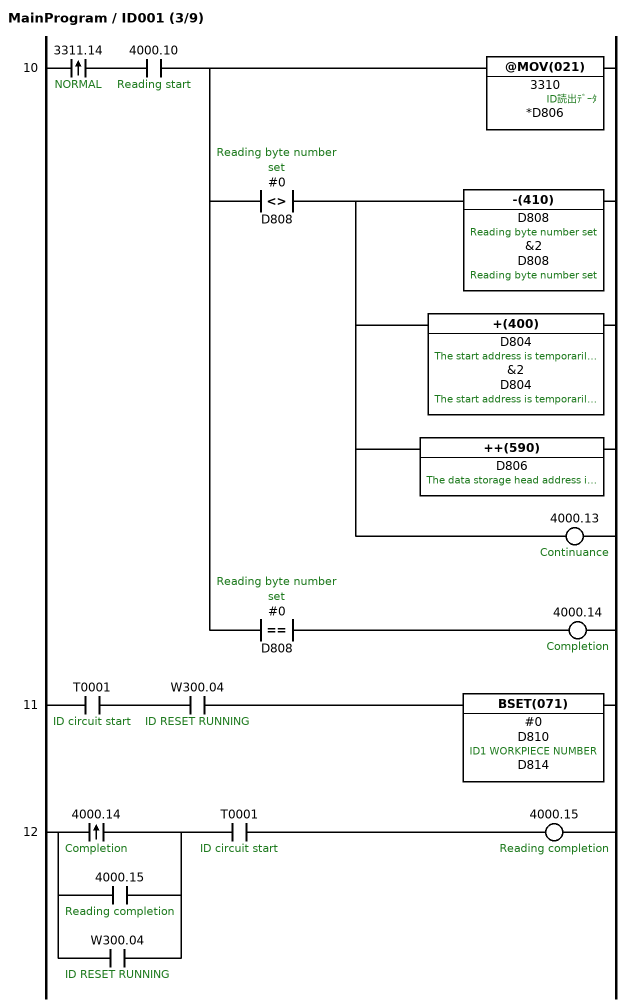
; [picture p24: MainProgram / ID001, rungs 10-12]
; rung 10
@LD 3311.14  ; NORMAL
AND 4000.10  ; Reading start
OUT TR0
@MOV(021) 3310 *D806  ; ID読出ﾃﾞｰﾀ
AND<>(305) #0 D808  ; Reading byte number set
-(410) D808 &2 D808  ; Reading byte number set
+(400) D804 &2 D804  ; The start address is temporarily memorized
++(590) D806  ; The data storage head address is memorized
OUT 4000.13  ; Continuance
LD TR0
AND=(300) #0 D808  ; Reading byte number set
OUT 4000.14  ; Completion
; rung 11
LD T0001  ; ID circuit start
AND W300.04  ; ID RESET RUNNING
BSET(071) #0 D810 D814  ; ID1 WORKPIECE NUMBER
; rung 12
@LD 4000.14  ; Completion
OR 4000.15  ; Reading completion
OR W300.04  ; ID RESET RUNNING
AND T0001  ; ID circuit start
OUT 4000.15  ; Reading completion

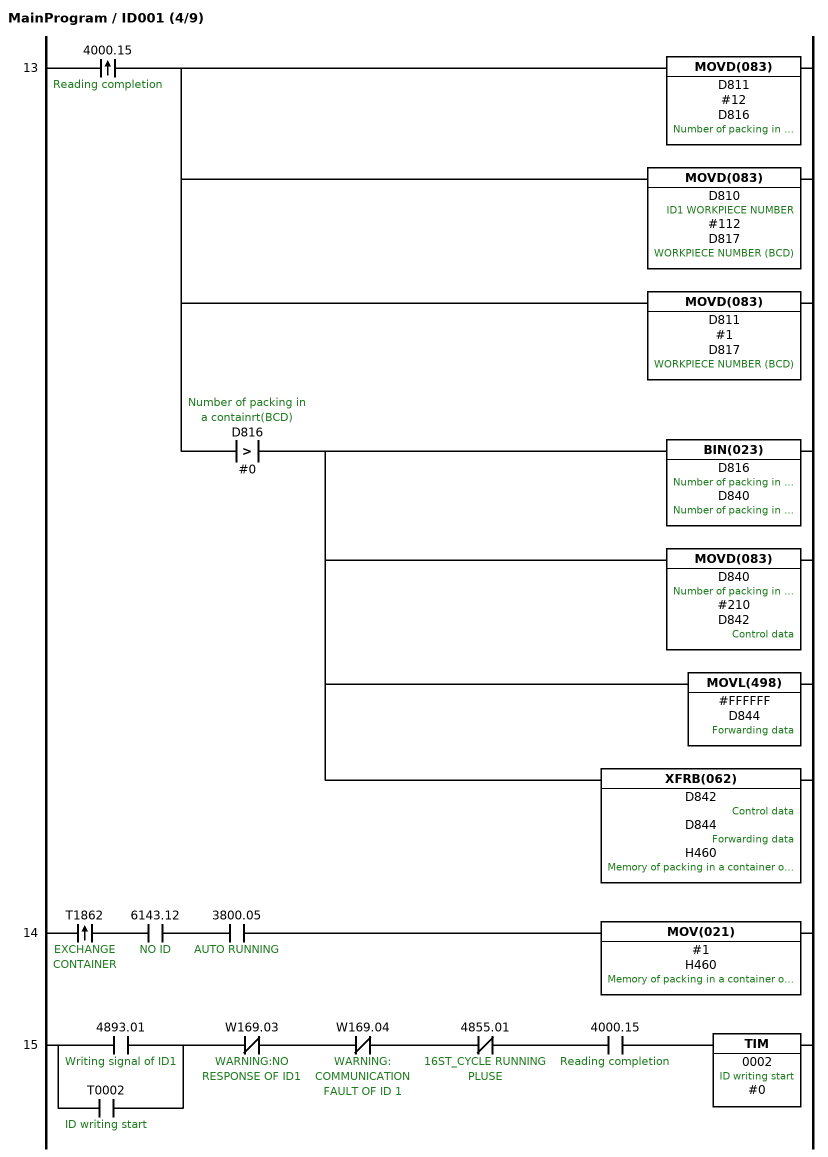
; rung 13
@LD 4000.15  ; Reading completion
MOVD(083) D811 #12 D816  ; Number of packing in a containrt(BCD)
MOVD(083) D810 #112 D817  ; ID1 WORKPIECE NUMBER, WORKPIECE NUMBER (BCD)
MOVD(083) D811 #1 D817  ; WORKPIECE NUMBER (BCD)
AND>(320) D816 #0  ; Number of packing in a containrt(BCD)
BIN(023) D816 D840  ; Number of packing in a containrt(BCD), Number of packing in a containrt(BIN)
MOVD(083) D840 #210 D842  ; Number of packing in a containrt(BIN), Control data
MOVL(498) #FFFFFF D844  ; Forwarding data
XFRB(062) D842 D844 H460  ; Control data, Forwarding data, Memory of packing in a container of lane 1 (exchange container)
; rung 14
@LD T1862  ; EXCHANGE CONTAINER
AND 6143.12  ; NO ID
AND 3800.05  ; AUTO RUNNING
MOV(021) #1 H460  ; Memory of packing in a container of lane 1 (exchange container)
; rung 15
LD 4893.01  ; Writing signal of ID1
OR T0002  ; ID writing start
ANDNOT W169.03  ; WARNING:NO RESPONSE OF ID1
ANDNOT W169.04  ; WARNING:COMMUNICATION FAULT OF ID 1
ANDNOT 4855.01  ; 16ST_CYCLE RUNNING PLUSE
AND 4000.15  ; Reading completion
TIM 0002 #0  ; ID writing start

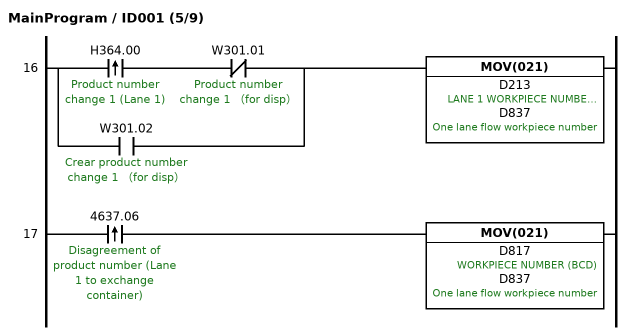
; rung 16
@LD H364.00  ; Product number change 1 (Lane 1)
ANDNOT W301.01  ; Product number change 1 （for disp）
OR W301.02  ; Crear product number change 1 （for disp）
MOV(021) D213 D837  ; LANE 1 WORKPIECE NUMBER DISPLAY, One lane flow workpiece number
; rung 17
@LD 4637.06  ; Disagreement of product number (Lane 1 to exchange container)
MOV(021) D817 D837  ; WORKPIECE NUMBER (BCD), One lane flow workpiece number

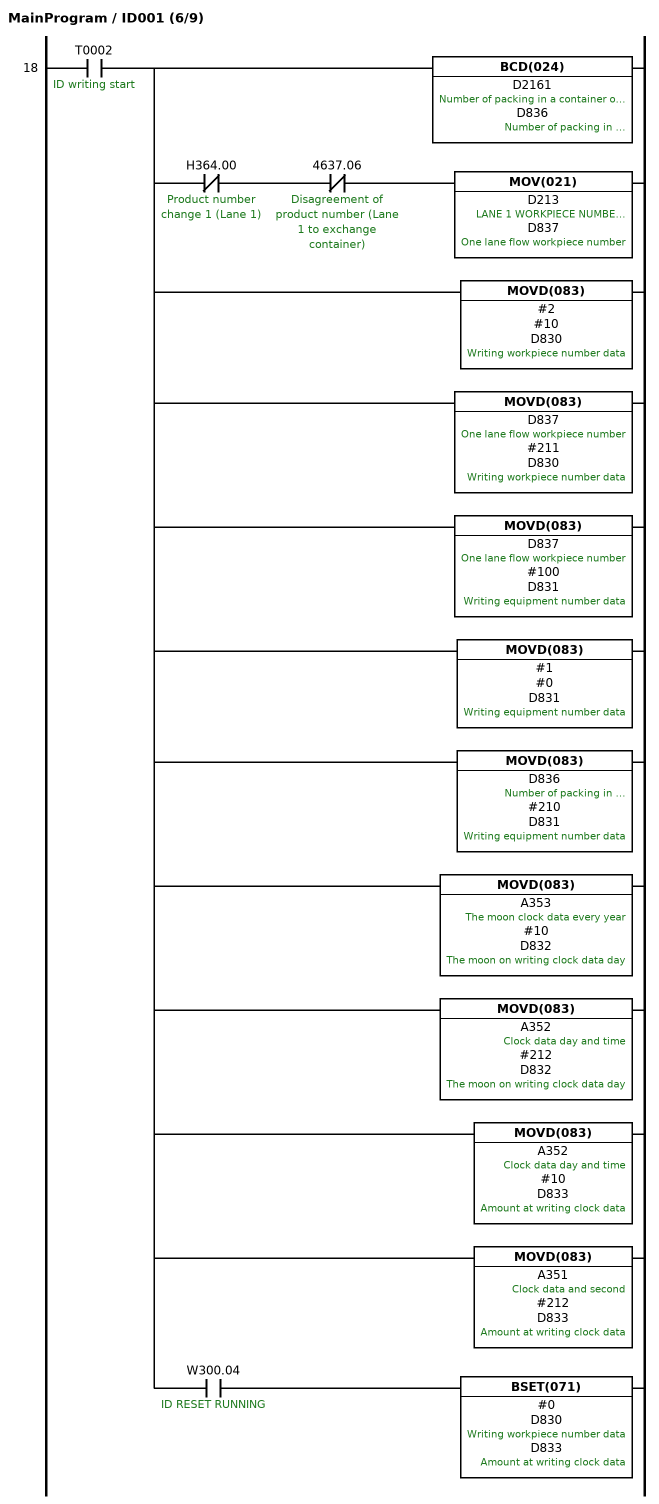
; rung 18
LD T0002  ; ID writing start
OUT TR0
BCD(024) D2161 D836  ; Number of packing in a container of lane 1 (exchange container)(BIN), Number of packing in a containrt(BCD)
ANDNOT H364.00  ; Product number change 1 (Lane 1)
ANDNOT 4637.06  ; Disagreement of product number (Lane 1 to exchange container)
MOV(021) D213 D837  ; LANE 1 WORKPIECE NUMBER DISPLAY, One lane flow workpiece number
LD TR0
MOVD(083) #2 #10 D830  ; Writing workpiece number data
MOVD(083) D837 #211 D830  ; One lane flow workpiece number, Writing workpiece number data
MOVD(083) D837 #100 D831  ; One lane flow workpiece number, Writing equipment number data
MOVD(083) #1 #0 D831  ; Writing equipment number data
MOVD(083) D836 #210 D831  ; Number of packing in a containrt(BCD), Writing equipment number data
MOVD(083) A353 #10 D832  ; The moon clock data every year, The moon on writing clock data day
MOVD(083) A352 #212 D832  ; Clock data day and time, The moon on writing clock data day
MOVD(083) A352 #10 D833  ; Clock data day and time, Amount at writing clock data
MOVD(083) A351 #212 D833  ; Clock data and second, Amount at writing clock data
AND W300.04  ; ID RESET RUNNING
BSET(071) #0 D830 D833  ; Writing workpiece number data, Amount at writing clock data

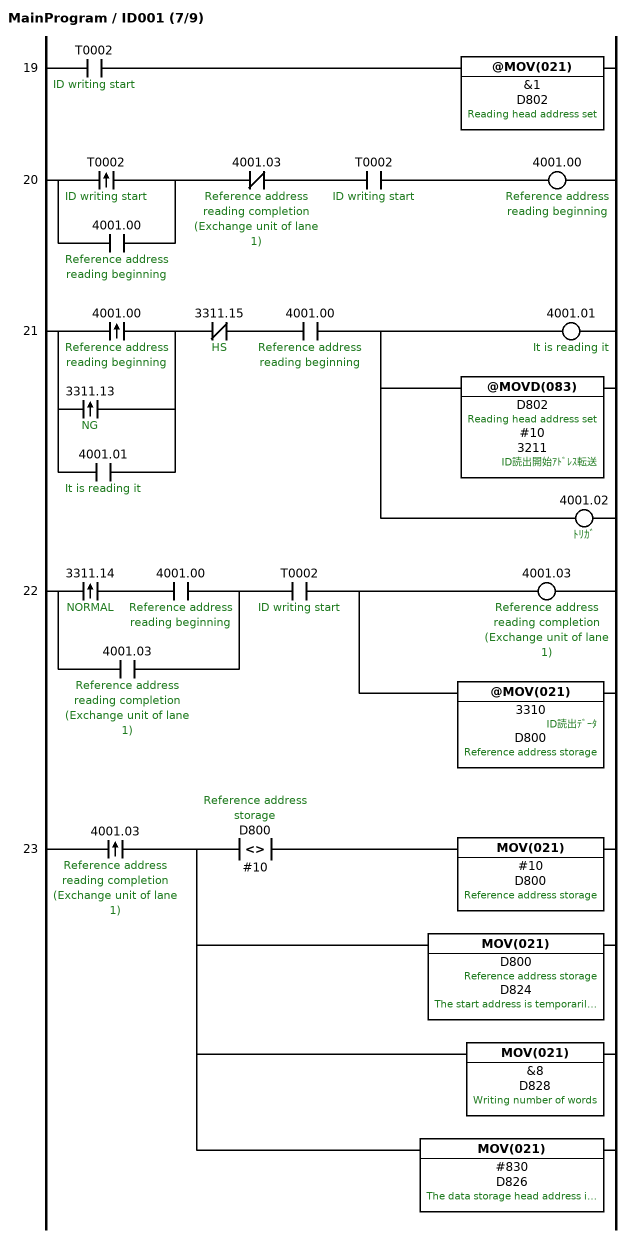
; rung 19
LD T0002  ; ID writing start
@MOV(021) &1 D802  ; Reading head address set
; rung 20
@LD T0002  ; ID writing start
OR 4001.00  ; Reference address reading beginning
ANDNOT 4001.03  ; Reference address reading completion (Exchange unit of lane 1)
AND T0002  ; ID writing start
OUT 4001.00  ; Reference address reading beginning
; rung 21
@LD 4001.00  ; Reference address reading beginning
@OR 3311.13  ; NG
OR 4001.01  ; It is reading it
ANDNOT 3311.15  ; HS
AND 4001.00  ; Reference address reading beginning
OUT 4001.01  ; It is reading it
@MOVD(083) D802 #10 3211  ; Reading head address set, ID読出開始ｱﾄﾞﾚｽ転送
OUT 4001.02  ; ﾄﾘｶﾞ
; rung 22
@LD 3311.14  ; NORMAL
AND 4001.00  ; Reference address reading beginning
OR 4001.03  ; Reference address reading completion (Exchange unit of lane 1)
AND T0002  ; ID writing start
OUT 4001.03  ; Reference address reading completion (Exchange unit of lane 1)
@MOV(021) 3310 D800  ; ID読出ﾃﾞｰﾀ, Reference address storage
; rung 23
@LD 4001.03  ; Reference address reading completion (Exchange unit of lane 1)
OUT TR0
AND<>(305) D800 #10  ; Reference address storage
MOV(021) #10 D800  ; Reference address storage
LD TR0
MOV(021) D800 D824  ; Reference address storage, The start address is temporarily memorized
MOV(021) &8 D828  ; Writing number of words
MOV(021) #830 D826  ; The data storage head address is memorized

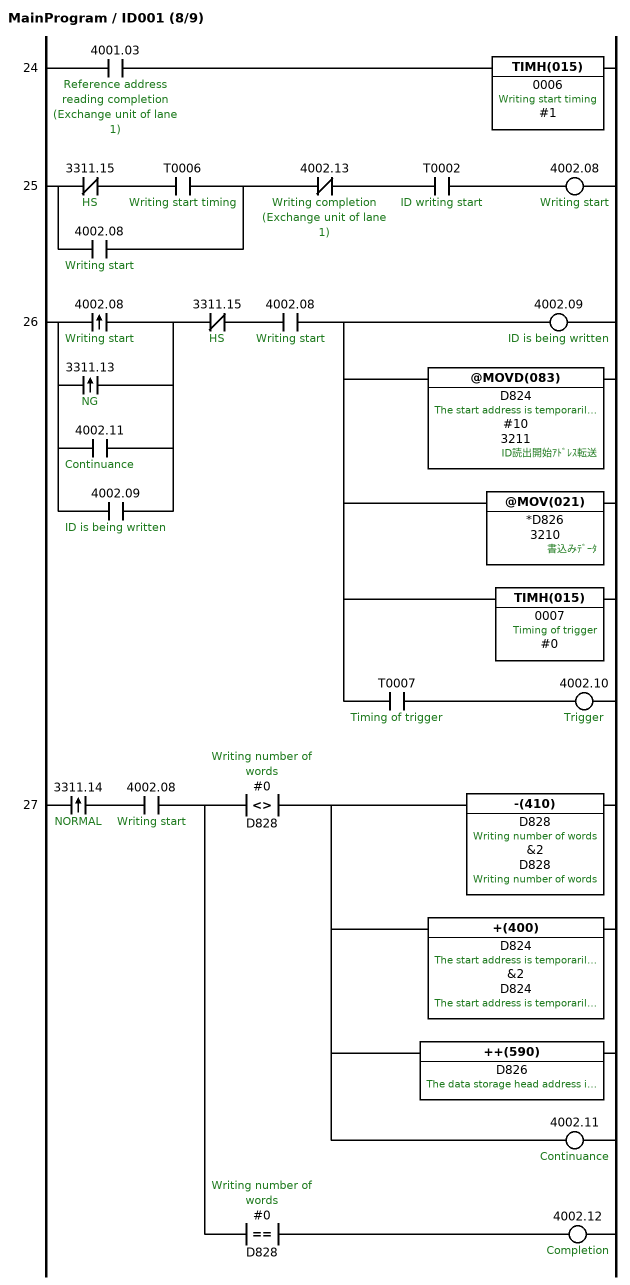
; rung 24
LD 4001.03  ; Reference address reading completion (Exchange unit of lane 1)
TIMH(015) 0006 #1  ; Writing start timing
; rung 25
LDNOT 3311.15  ; HS
AND T0006  ; Writing start timing
OR 4002.08  ; Writing start
ANDNOT 4002.13  ; Writing completion (Exchange unit of lane 1)
AND T0002  ; ID writing start
OUT 4002.08  ; Writing start
; rung 26
@LD 4002.08  ; Writing start
@OR 3311.13  ; NG
OR 4002.11  ; Continuance
OR 4002.09  ; ID is being written
ANDNOT 3311.15  ; HS
AND 4002.08  ; Writing start
OUT 4002.09  ; ID is being written
@MOVD(083) D824 #10 3211  ; The start address is temporarily memorized, ID読出開始ｱﾄﾞﾚｽ転送
@MOV(021) *D826 3210  ; 書込みﾃﾞｰﾀ
TIMH(015) 0007 #0  ; Timing of trigger
AND T0007  ; Timing of trigger
OUT 4002.10  ; Trigger
; rung 27
@LD 3311.14  ; NORMAL
AND 4002.08  ; Writing start
OUT TR0
AND<>(305) #0 D828  ; Writing number of words
-(410) D828 &2 D828  ; Writing number of words
+(400) D824 &2 D824  ; The start address is temporarily memorized
++(590) D826  ; The data storage head address is memorized
OUT 4002.11  ; Continuance
LD TR0
AND=(300) #0 D828  ; Writing number of words
OUT 4002.12  ; Completion

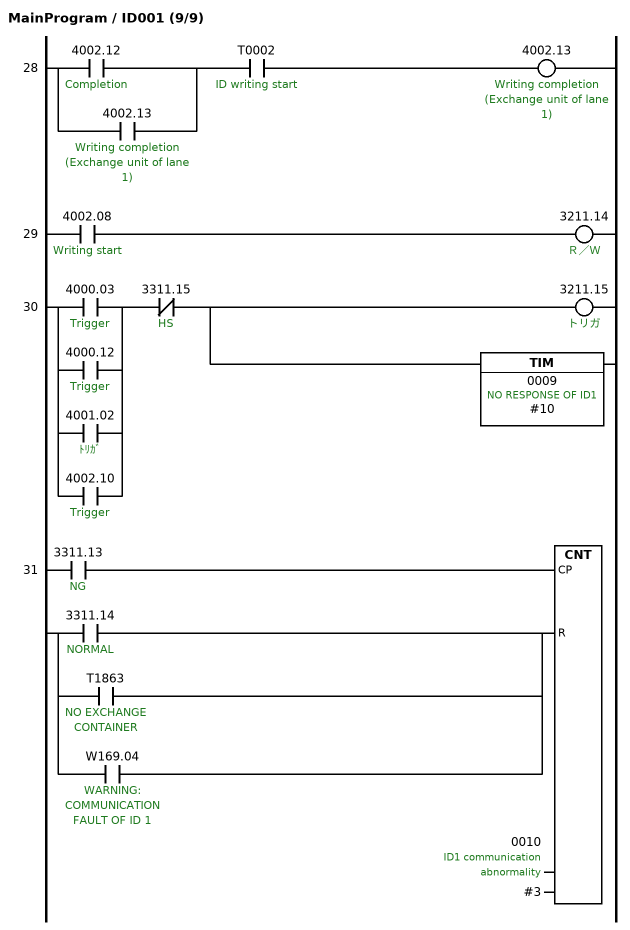
; rung 28
LD 4002.12  ; Completion
OR 4002.13  ; Writing completion (Exchange unit of lane 1)
AND T0002  ; ID writing start
OUT 4002.13  ; Writing completion (Exchange unit of lane 1)
; rung 29
LD 4002.08  ; Writing start
OUT 3211.14  ; Ｒ／Ｗ
; rung 30
LD 4000.03  ; Trigger
OR 4000.12  ; Trigger
OR 4001.02  ; ﾄﾘｶﾞ
OR 4002.10  ; Trigger
ANDNOT 3311.15  ; HS
OUT 3211.15  ; トリガ
TIM 0009 #10  ; NO RESPONSE OF ID1
; rung 31
LD 3311.13  ; NG
LD 3311.14  ; NORMAL
OR T1863  ; NO EXCHANGE CONTAINER
OR W169.04  ; WARNING:COMMUNICATION FAULT OF ID 1
CNT 0010 #3  ; ID1 communication abnormality

### Section ID002

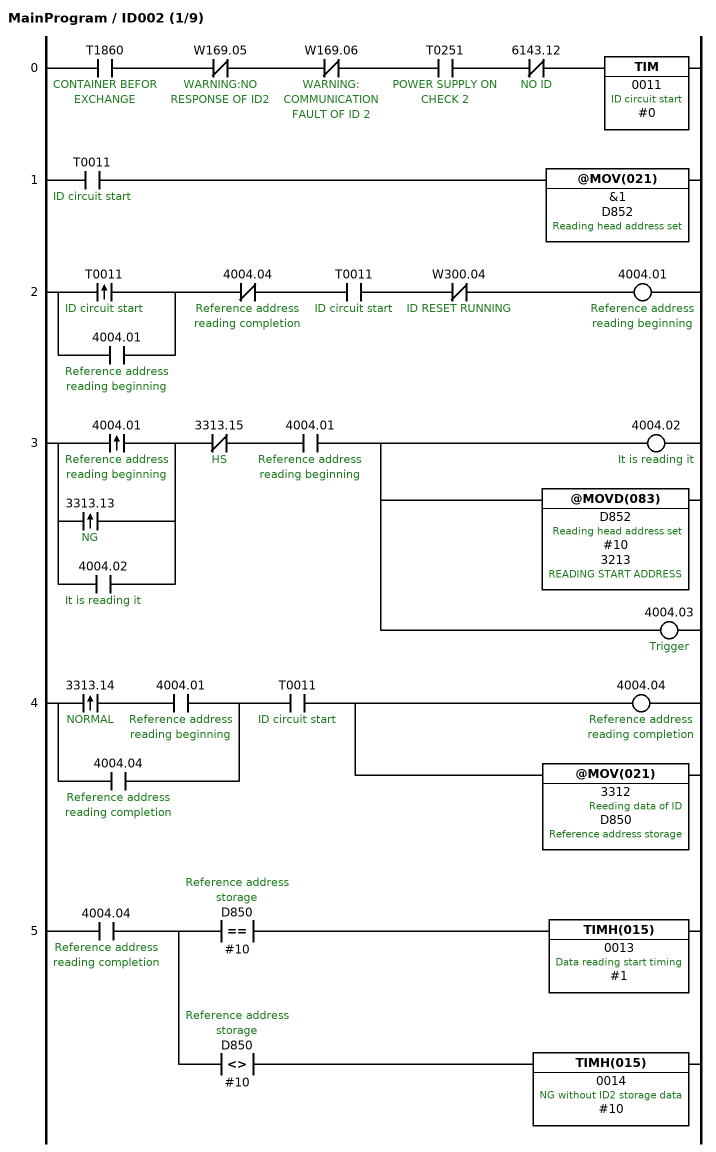
; rung 0
LD T1860  ; CONTAINER BEFOR EXCHANGE
ANDNOT W169.05  ; WARNING:NO RESPONSE OF ID2
ANDNOT W169.06  ; WARNING:COMMUNICATION FAULT OF ID 2
AND T0251  ; POWER SUPPLY ON CHECK 2
ANDNOT 6143.12  ; NO ID
TIM 0011 #0  ; ID circuit start
; rung 1
LD T0011  ; ID circuit start
@MOV(021) &1 D852  ; Reading head address set
; rung 2
@LD T0011  ; ID circuit start
OR 4004.01  ; Reference address reading beginning
ANDNOT 4004.04  ; Reference address reading completion
AND T0011  ; ID circuit start
ANDNOT W300.04  ; ID RESET RUNNING
OUT 4004.01  ; Reference address reading beginning
; rung 3
@LD 4004.01  ; Reference address reading beginning
@OR 3313.13  ; NG
OR 4004.02  ; It is reading it
ANDNOT 3313.15  ; HS
AND 4004.01  ; Reference address reading beginning
OUT 4004.02  ; It is reading it
@MOVD(083) D852 #10 3213  ; Reading head address set, READING START ADDRESS
OUT 4004.03  ; Trigger
; rung 4
@LD 3313.14  ; NORMAL
AND 4004.01  ; Reference address reading beginning
OR 4004.04  ; Reference address reading completion
AND T0011  ; ID circuit start
OUT 4004.04  ; Reference address reading completion
@MOV(021) 3312 D850  ; Reeding data of ID, Reference address storage
; rung 5
LD 4004.04  ; Reference address reading completion
OUT TR0
AND=(300) D850 #10  ; Reference address storage
TIMH(015) 0013 #1  ; Data reading start timing
LD TR0
AND<>(305) D850 #10  ; Reference address storage
TIMH(015) 0014 #10  ; NG without ID2 storage data

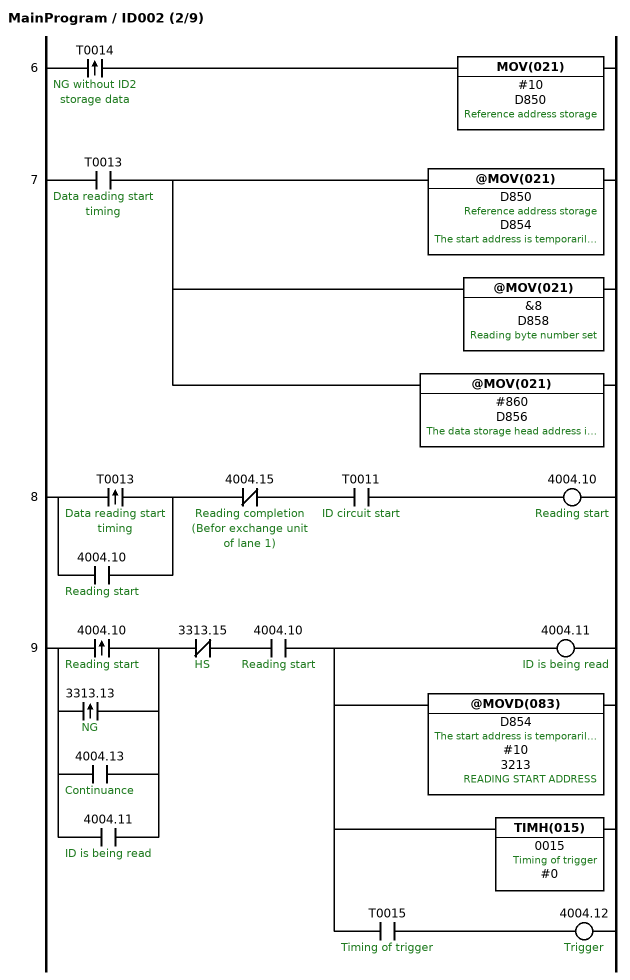
; rung 6
@LD T0014  ; NG without ID2 storage data
MOV(021) #10 D850  ; Reference address storage
; rung 7
LD T0013  ; Data reading start timing
@MOV(021) D850 D854  ; Reference address storage, The start address is temporarily memorized
@MOV(021) &8 D858  ; Reading byte number set
@MOV(021) #860 D856  ; The data storage head address is memorized
; rung 8
@LD T0013  ; Data reading start timing
OR 4004.10  ; Reading start
ANDNOT 4004.15  ; Reading completion (Befor exchange unit of lane 1)
AND T0011  ; ID circuit start
OUT 4004.10  ; Reading start
; rung 9
@LD 4004.10  ; Reading start
@OR 3313.13  ; NG
OR 4004.13  ; Continuance
OR 4004.11  ; ID is being read
ANDNOT 3313.15  ; HS
AND 4004.10  ; Reading start
OUT 4004.11  ; ID is being read
@MOVD(083) D854 #10 3213  ; The start address is temporarily memorized, READING START ADDRESS
TIMH(015) 0015 #0  ; Timing of trigger
AND T0015  ; Timing of trigger
OUT 4004.12  ; Trigger

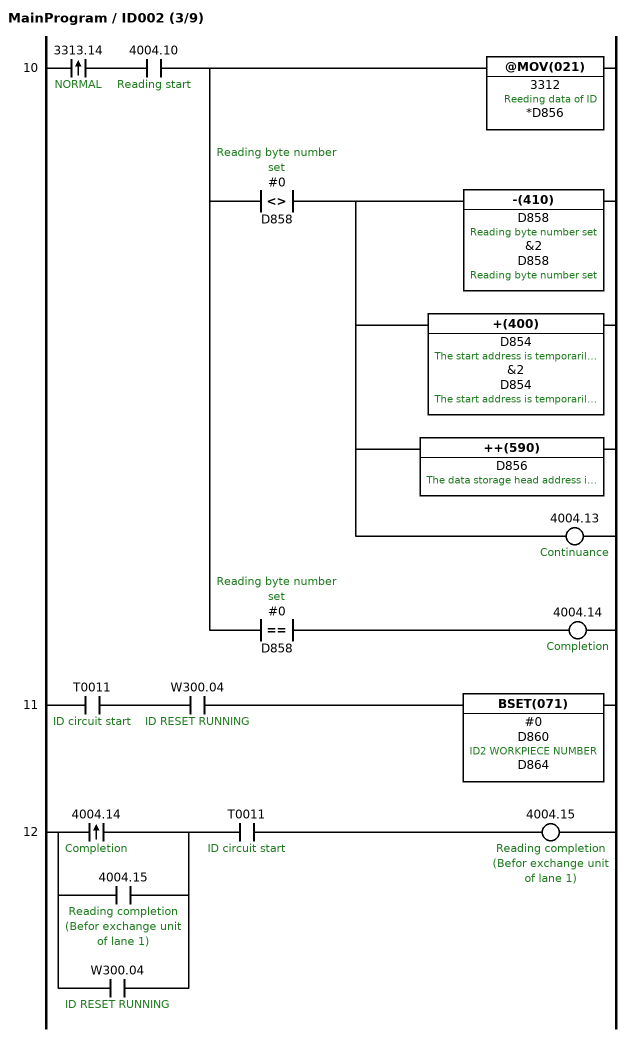
; rung 10
@LD 3313.14  ; NORMAL
AND 4004.10  ; Reading start
OUT TR0
@MOV(021) 3312 *D856  ; Reeding data of ID
AND<>(305) #0 D858  ; Reading byte number set
-(410) D858 &2 D858  ; Reading byte number set
+(400) D854 &2 D854  ; The start address is temporarily memorized
++(590) D856  ; The data storage head address is memorized
OUT 4004.13  ; Continuance
LD TR0
AND=(300) #0 D858  ; Reading byte number set
OUT 4004.14  ; Completion
; rung 11
LD T0011  ; ID circuit start
AND W300.04  ; ID RESET RUNNING
BSET(071) #0 D860 D864  ; ID2 WORKPIECE NUMBER
; rung 12
@LD 4004.14  ; Completion
OR 4004.15  ; Reading completion (Befor exchange unit of lane 1)
OR W300.04  ; ID RESET RUNNING
AND T0011  ; ID circuit start
OUT 4004.15  ; Reading completion (Befor exchange unit of lane 1)

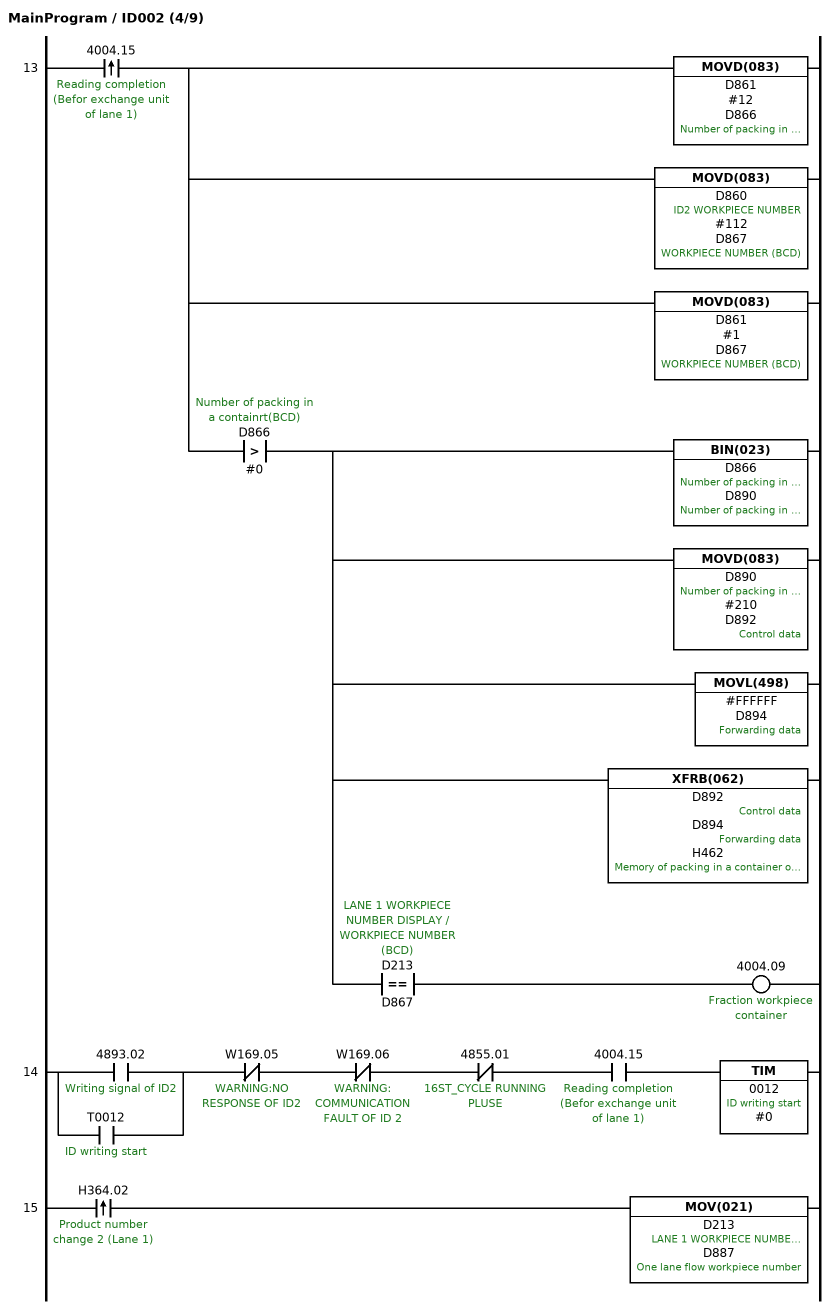
; rung 13
@LD 4004.15  ; Reading completion (Befor exchange unit of lane 1)
MOVD(083) D861 #12 D866  ; Number of packing in a containrt(BCD)
MOVD(083) D860 #112 D867  ; ID2 WORKPIECE NUMBER, WORKPIECE NUMBER (BCD)
MOVD(083) D861 #1 D867  ; WORKPIECE NUMBER (BCD)
AND>(320) D866 #0  ; Number of packing in a containrt(BCD)
BIN(023) D866 D890  ; Number of packing in a containrt(BCD), Number of packing in a containrt(BIN)
MOVD(083) D890 #210 D892  ; Number of packing in a containrt(BIN), Control data
MOVL(498) #FFFFFF D894  ; Forwarding data
XFRB(062) D892 D894 H462  ; Control data, Forwarding data, Memory of packing in a container of lane 1 (container befor exchange)
AND=(300) D213 D867  ; LANE 1 WORKPIECE NUMBER DISPLAY, WORKPIECE NUMBER (BCD)
OUT 4004.09  ; Fraction workpiece container
; rung 14
LD 4893.02  ; Writing signal of ID2
OR T0012  ; ID writing start
ANDNOT W169.05  ; WARNING:NO RESPONSE OF ID2
ANDNOT W169.06  ; WARNING:COMMUNICATION FAULT OF ID 2
ANDNOT 4855.01  ; 16ST_CYCLE RUNNING PLUSE
AND 4004.15  ; Reading completion (Befor exchange unit of lane 1)
TIM 0012 #0  ; ID writing start
; rung 15
@LD H364.02  ; Product number change 2 (Lane 1)
MOV(021) D213 D887  ; LANE 1 WORKPIECE NUMBER DISPLAY, One lane flow workpiece number

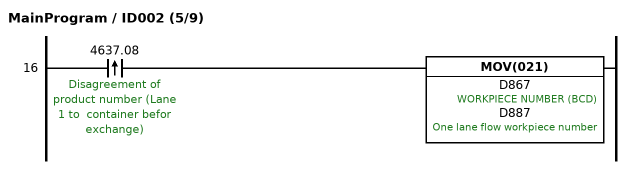
; rung 16
@LD 4637.08  ; Disagreement of product number (Lane 1 to  container befor exchange)
MOV(021) D867 D887  ; WORKPIECE NUMBER (BCD), One lane flow workpiece number

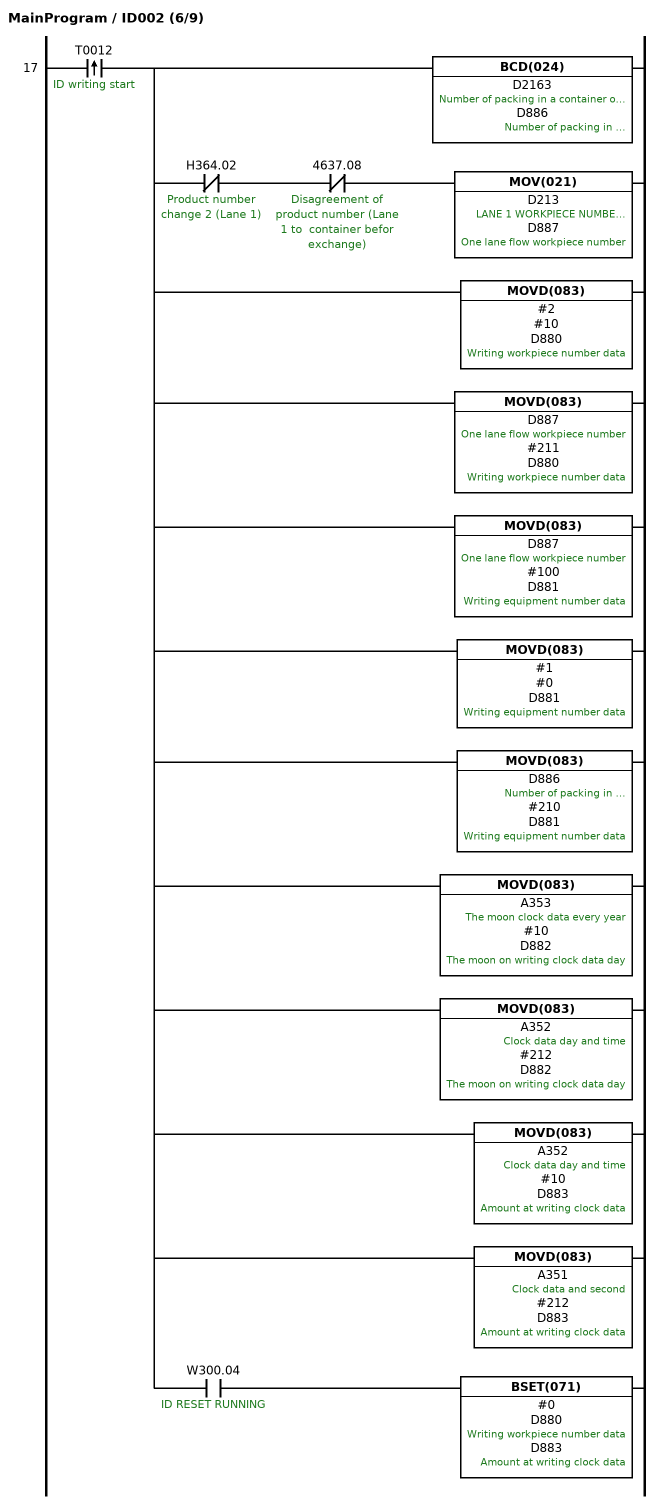
; rung 17
@LD T0012  ; ID writing start
OUT TR0
BCD(024) D2163 D886  ; Number of packing in a container of lane 1 (container before exchange)(BIN), Number of packing in a containrt(BCD)
ANDNOT H364.02  ; Product number change 2 (Lane 1)
ANDNOT 4637.08  ; Disagreement of product number (Lane 1 to  container befor exchange)
MOV(021) D213 D887  ; LANE 1 WORKPIECE NUMBER DISPLAY, One lane flow workpiece number
LD TR0
MOVD(083) #2 #10 D880  ; Writing workpiece number data
MOVD(083) D887 #211 D880  ; One lane flow workpiece number, Writing workpiece number data
MOVD(083) D887 #100 D881  ; One lane flow workpiece number, Writing equipment number data
MOVD(083) #1 #0 D881  ; Writing equipment number data
MOVD(083) D886 #210 D881  ; Number of packing in a containrt(BCD), Writing equipment number data
MOVD(083) A353 #10 D882  ; The moon clock data every year, The moon on writing clock data day
MOVD(083) A352 #212 D882  ; Clock data day and time, The moon on writing clock data day
MOVD(083) A352 #10 D883  ; Clock data day and time, Amount at writing clock data
MOVD(083) A351 #212 D883  ; Clock data and second, Amount at writing clock data
AND W300.04  ; ID RESET RUNNING
BSET(071) #0 D880 D883  ; Writing workpiece number data, Amount at writing clock data

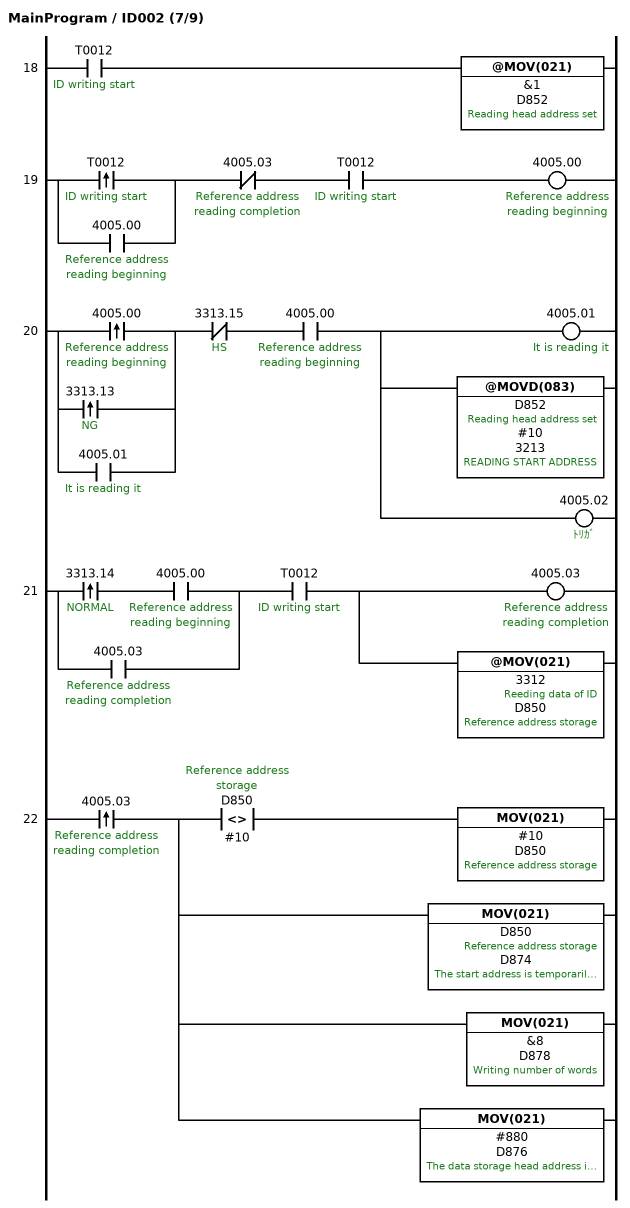
; rung 18
LD T0012  ; ID writing start
@MOV(021) &1 D852  ; Reading head address set
; rung 19
@LD T0012  ; ID writing start
OR 4005.00  ; Reference address reading beginning
ANDNOT 4005.03  ; Reference address reading completion
AND T0012  ; ID writing start
OUT 4005.00  ; Reference address reading beginning
; rung 20
@LD 4005.00  ; Reference address reading beginning
@OR 3313.13  ; NG
OR 4005.01  ; It is reading it
ANDNOT 3313.15  ; HS
AND 4005.00  ; Reference address reading beginning
OUT 4005.01  ; It is reading it
@MOVD(083) D852 #10 3213  ; Reading head address set, READING START ADDRESS
OUT 4005.02  ; ﾄﾘｶﾞ
; rung 21
@LD 3313.14  ; NORMAL
AND 4005.00  ; Reference address reading beginning
OR 4005.03  ; Reference address reading completion
AND T0012  ; ID writing start
OUT 4005.03  ; Reference address reading completion
@MOV(021) 3312 D850  ; Reeding data of ID, Reference address storage
; rung 22
@LD 4005.03  ; Reference address reading completion
OUT TR0
AND<>(305) D850 #10  ; Reference address storage
MOV(021) #10 D850  ; Reference address storage
LD TR0
MOV(021) D850 D874  ; Reference address storage, The start address is temporarily memorized
MOV(021) &8 D878  ; Writing number of words
MOV(021) #880 D876  ; The data storage head address is memorized

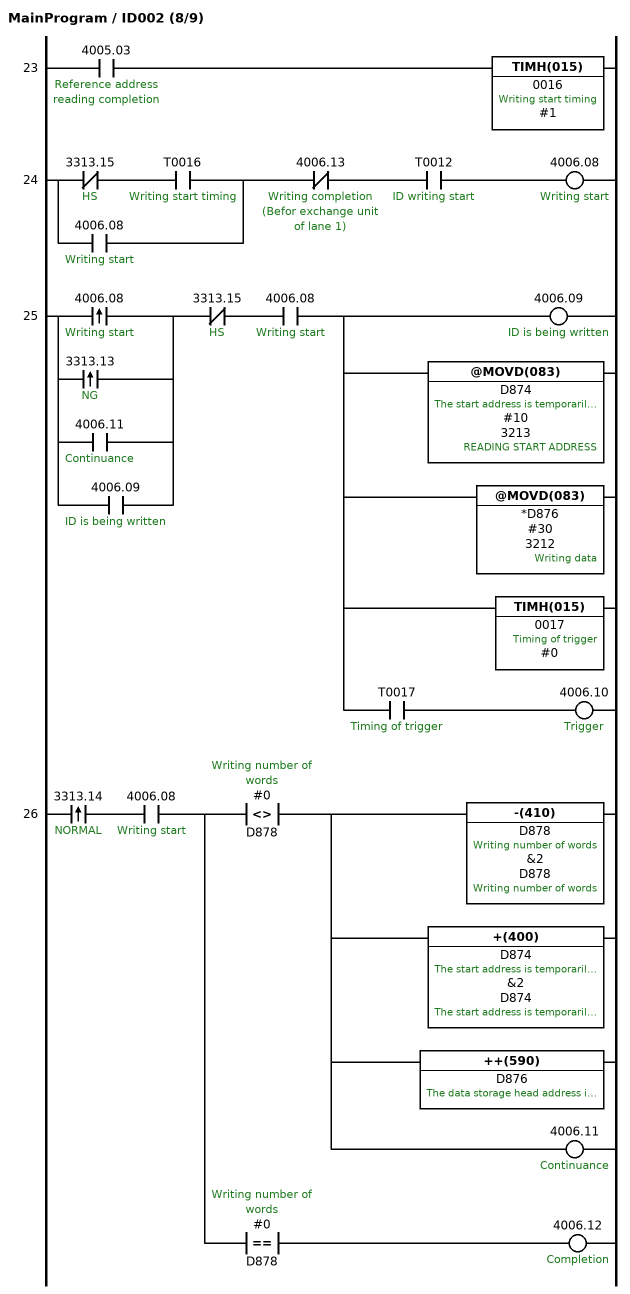
; rung 23
LD 4005.03  ; Reference address reading completion
TIMH(015) 0016 #1  ; Writing start timing
; rung 24
LDNOT 3313.15  ; HS
AND T0016  ; Writing start timing
OR 4006.08  ; Writing start
ANDNOT 4006.13  ; Writing completion (Befor exchange unit of lane 1)
AND T0012  ; ID writing start
OUT 4006.08  ; Writing start
; rung 25
@LD 4006.08  ; Writing start
@OR 3313.13  ; NG
OR 4006.11  ; Continuance
OR 4006.09  ; ID is being written
ANDNOT 3313.15  ; HS
AND 4006.08  ; Writing start
OUT 4006.09  ; ID is being written
@MOVD(083) D874 #10 3213  ; The start address is temporarily memorized, READING START ADDRESS
@MOVD(083) *D876 #30 3212  ; Writing data
TIMH(015) 0017 #0  ; Timing of trigger
AND T0017  ; Timing of trigger
OUT 4006.10  ; Trigger
; rung 26
@LD 3313.14  ; NORMAL
AND 4006.08  ; Writing start
OUT TR0
AND<>(305) #0 D878  ; Writing number of words
-(410) D878 &2 D878  ; Writing number of words
+(400) D874 &2 D874  ; The start address is temporarily memorized
++(590) D876  ; The data storage head address is memorized
OUT 4006.11  ; Continuance
LD TR0
AND=(300) #0 D878  ; Writing number of words
OUT 4006.12  ; Completion

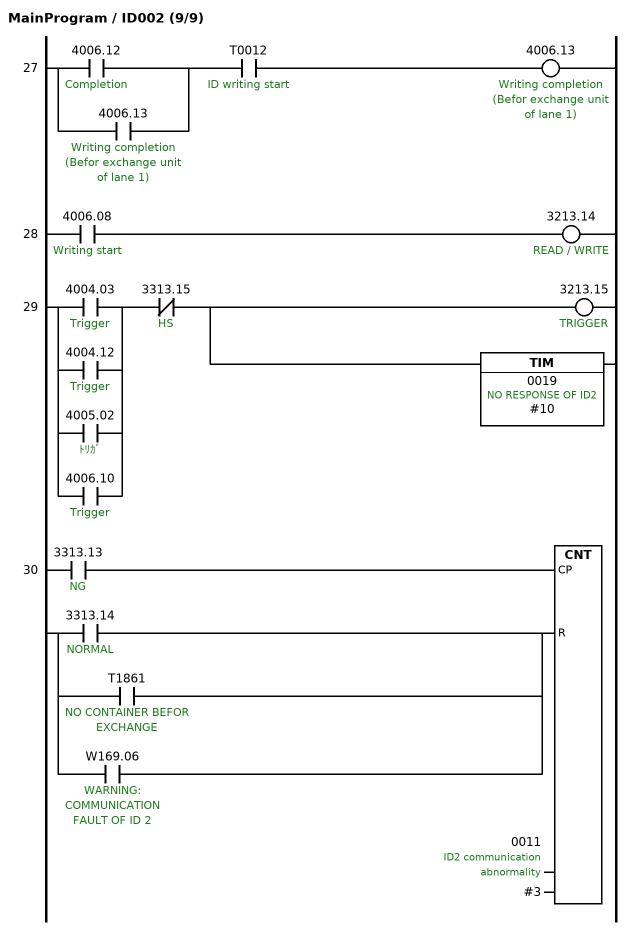
; rung 27
LD 4006.12  ; Completion
OR 4006.13  ; Writing completion (Befor exchange unit of lane 1)
AND T0012  ; ID writing start
OUT 4006.13  ; Writing completion (Befor exchange unit of lane 1)
; rung 28
LD 4006.08  ; Writing start
OUT 3213.14  ; READ / WRITE
; rung 29
LD 4004.03  ; Trigger
OR 4004.12  ; Trigger
OR 4005.02  ; ﾄﾘｶﾞ
OR 4006.10  ; Trigger
ANDNOT 3313.15  ; HS
OUT 3213.15  ; TRIGGER
TIM 0019 #10  ; NO RESPONSE OF ID2
; rung 30
LD 3313.13  ; NG
LD 3313.14  ; NORMAL
OR T1861  ; NO CONTAINER BEFOR EXCHANGE
OR W169.06  ; WARNING:COMMUNICATION FAULT OF ID 2
CNT 0011 #3  ; ID2 communication abnormality

### Section ID003

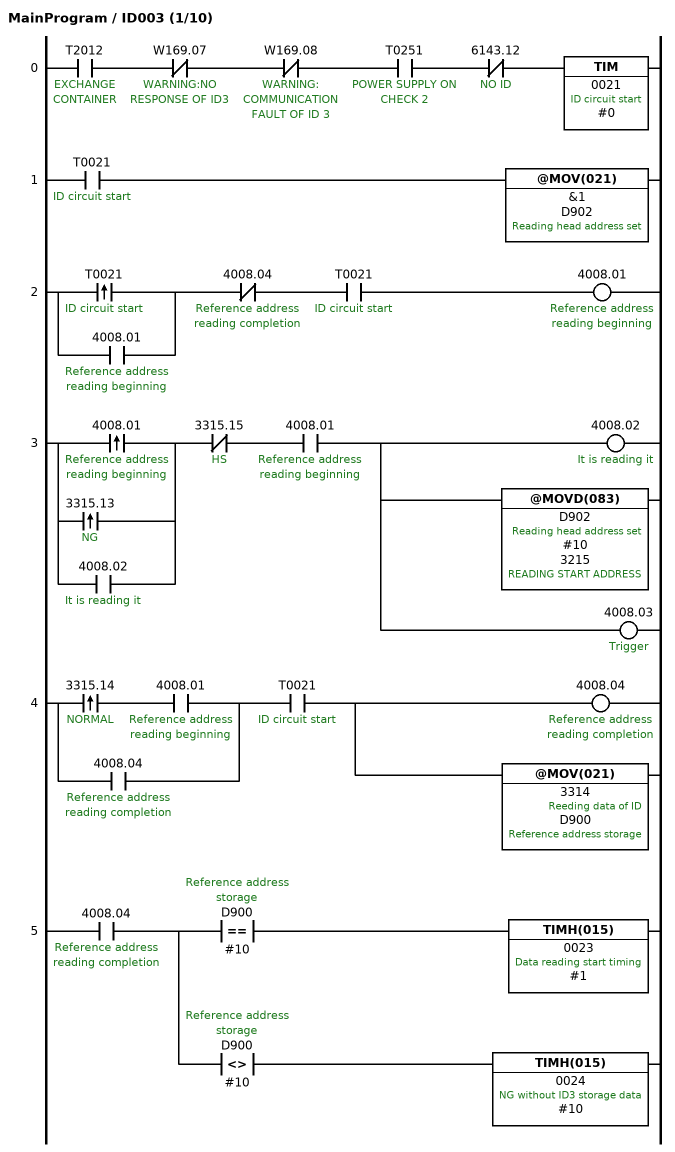
; rung 0
LD T2012  ; EXCHANGE CONTAINER
ANDNOT W169.07  ; WARNING:NO RESPONSE OF ID3
ANDNOT W169.08  ; WARNING:COMMUNICATION FAULT OF ID 3
AND T0251  ; POWER SUPPLY ON CHECK 2
ANDNOT 6143.12  ; NO ID
TIM 0021 #0  ; ID circuit start
; rung 1
LD T0021  ; ID circuit start
@MOV(021) &1 D902  ; Reading head address set
; rung 2
@LD T0021  ; ID circuit start
OR 4008.01  ; Reference address reading beginning
ANDNOT 4008.04  ; Reference address reading completion
AND T0021  ; ID circuit start
OUT 4008.01  ; Reference address reading beginning
; rung 3
@LD 4008.01  ; Reference address reading beginning
@OR 3315.13  ; NG
OR 4008.02  ; It is reading it
ANDNOT 3315.15  ; HS
AND 4008.01  ; Reference address reading beginning
OUT 4008.02  ; It is reading it
@MOVD(083) D902 #10 3215  ; Reading head address set, READING START ADDRESS
OUT 4008.03  ; Trigger
; rung 4
@LD 3315.14  ; NORMAL
AND 4008.01  ; Reference address reading beginning
OR 4008.04  ; Reference address reading completion
AND T0021  ; ID circuit start
OUT 4008.04  ; Reference address reading completion
@MOV(021) 3314 D900  ; Reeding data of ID, Reference address storage
; rung 5
LD 4008.04  ; Reference address reading completion
OUT TR0
AND=(300) D900 #10  ; Reference address storage
TIMH(015) 0023 #1  ; Data reading start timing
LD TR0
AND<>(305) D900 #10  ; Reference address storage
TIMH(015) 0024 #10  ; NG without ID3 storage data

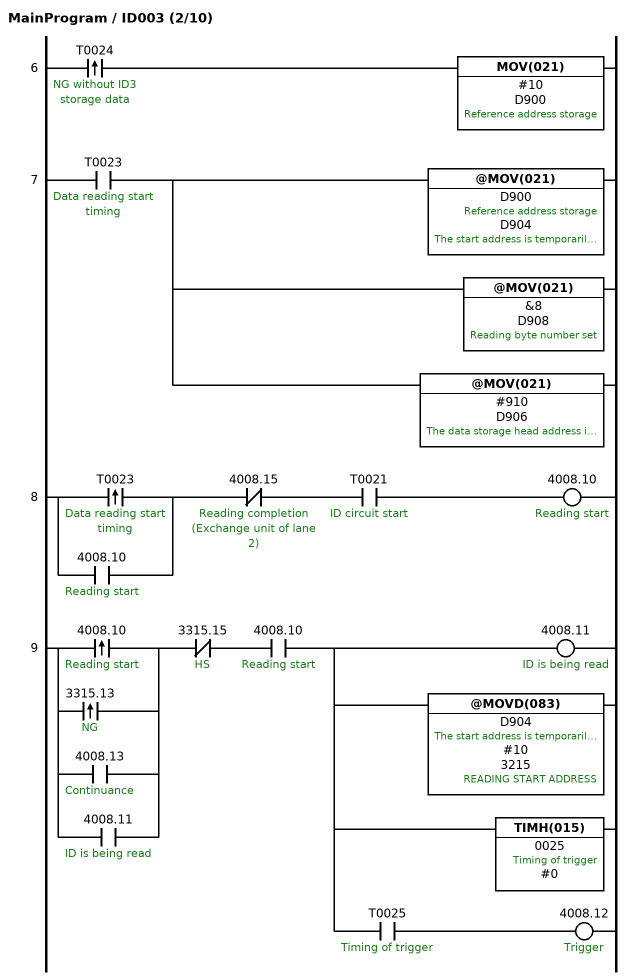
; rung 6
@LD T0024  ; NG without ID3 storage data
MOV(021) #10 D900  ; Reference address storage
; rung 7
LD T0023  ; Data reading start timing
@MOV(021) D900 D904  ; Reference address storage, The start address is temporarily memorized
@MOV(021) &8 D908  ; Reading byte number set
@MOV(021) #910 D906  ; The data storage head address is memorized
; rung 8
@LD T0023  ; Data reading start timing
OR 4008.10  ; Reading start
ANDNOT 4008.15  ; Reading completion (Exchange unit of lane 2)
AND T0021  ; ID circuit start
OUT 4008.10  ; Reading start
; rung 9
@LD 4008.10  ; Reading start
@OR 3315.13  ; NG
OR 4008.13  ; Continuance
OR 4008.11  ; ID is being read
ANDNOT 3315.15  ; HS
AND 4008.10  ; Reading start
OUT 4008.11  ; ID is being read
@MOVD(083) D904 #10 3215  ; The start address is temporarily memorized, READING START ADDRESS
TIMH(015) 0025 #0  ; Timing of trigger
AND T0025  ; Timing of trigger
OUT 4008.12  ; Trigger

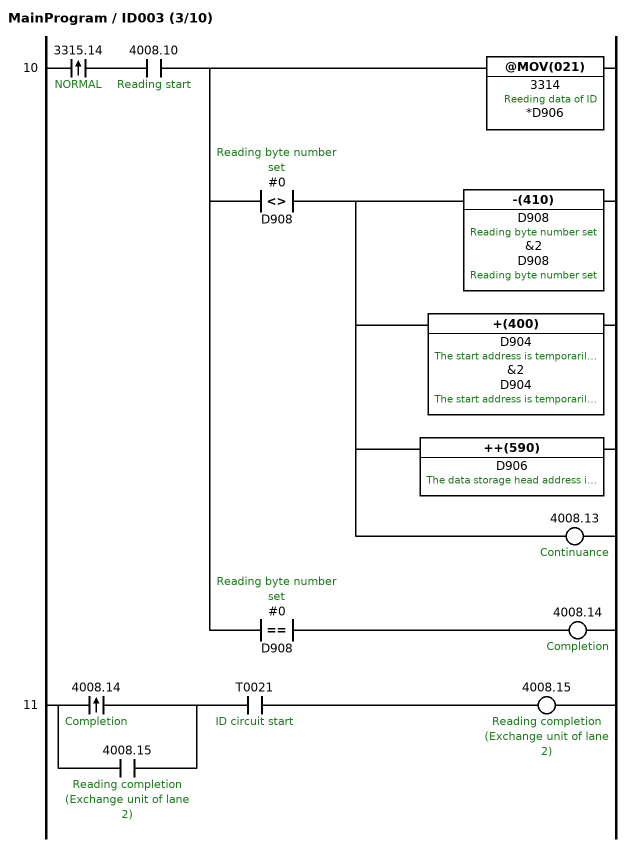
; rung 10
@LD 3315.14  ; NORMAL
AND 4008.10  ; Reading start
OUT TR0
@MOV(021) 3314 *D906  ; Reeding data of ID
AND<>(305) #0 D908  ; Reading byte number set
-(410) D908 &2 D908  ; Reading byte number set
+(400) D904 &2 D904  ; The start address is temporarily memorized
++(590) D906  ; The data storage head address is memorized
OUT 4008.13  ; Continuance
LD TR0
AND=(300) #0 D908  ; Reading byte number set
OUT 4008.14  ; Completion
; rung 11
@LD 4008.14  ; Completion
OR 4008.15  ; Reading completion (Exchange unit of lane 2)
AND T0021  ; ID circuit start
OUT 4008.15  ; Reading completion (Exchange unit of lane 2)

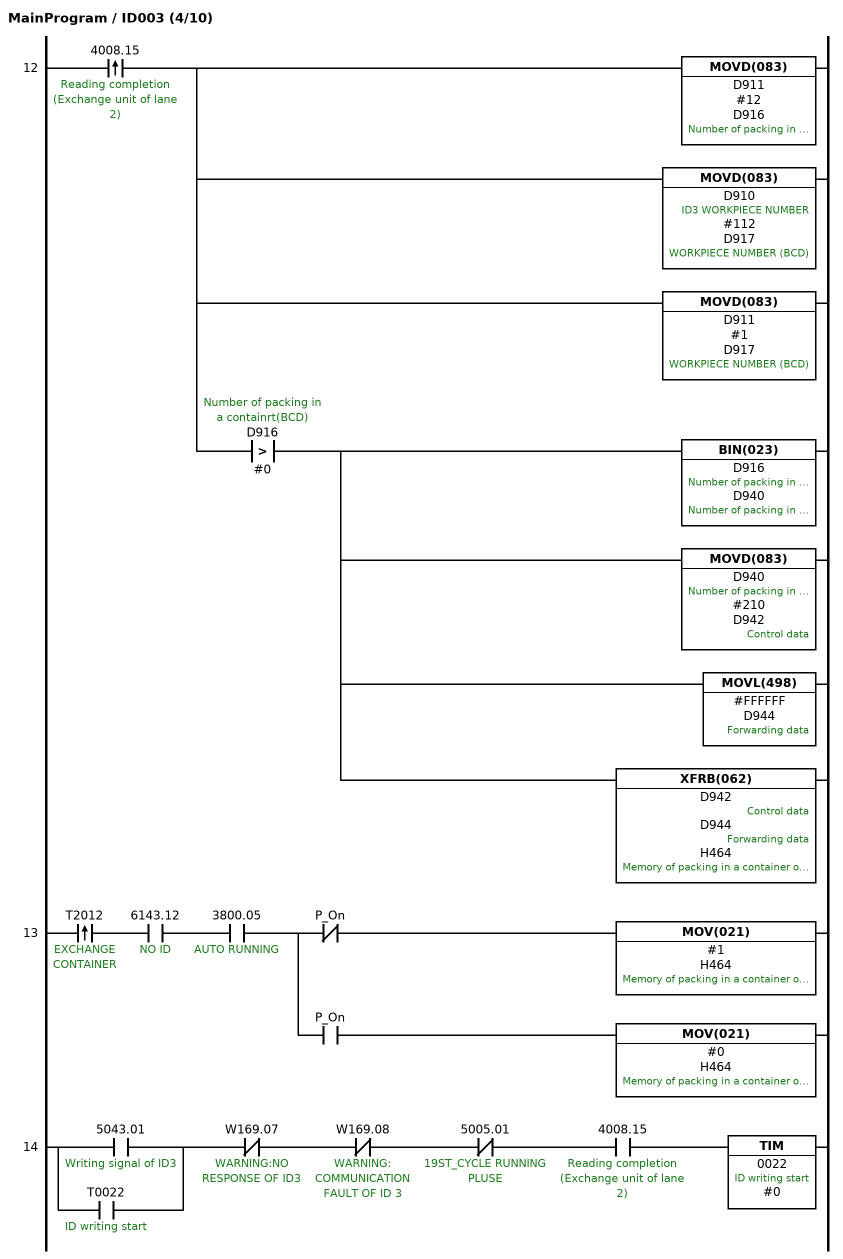
; rung 12
@LD 4008.15  ; Reading completion (Exchange unit of lane 2)
MOVD(083) D911 #12 D916  ; Number of packing in a containrt(BCD)
MOVD(083) D910 #112 D917  ; ID3 WORKPIECE NUMBER, WORKPIECE NUMBER (BCD)
MOVD(083) D911 #1 D917  ; WORKPIECE NUMBER (BCD)
AND>(320) D916 #0  ; Number of packing in a containrt(BCD)
BIN(023) D916 D940  ; Number of packing in a containrt(BCD), Number of packing in a containrt(BIN)
MOVD(083) D940 #210 D942  ; Number of packing in a containrt(BIN), Control data
MOVL(498) #FFFFFF D944  ; Forwarding data
XFRB(062) D942 D944 H464  ; Control data, Forwarding data, Memory of packing in a container of lane 2 (exchange container)
; rung 13
@LD T2012  ; EXCHANGE CONTAINER
AND 6143.12  ; NO ID
AND 3800.05  ; AUTO RUNNING
OUT TR0
ANDNOT P_On
MOV(021) #1 H464  ; Memory of packing in a container of lane 2 (exchange container)
LD TR0
AND P_On
MOV(021) #0 H464  ; Memory of packing in a container of lane 2 (exchange container)
; rung 14
LD 5043.01  ; Writing signal of ID3
OR T0022  ; ID writing start
ANDNOT W169.07  ; WARNING:NO RESPONSE OF ID3
ANDNOT W169.08  ; WARNING:COMMUNICATION FAULT OF ID 3
ANDNOT 5005.01  ; 19ST_CYCLE RUNNING PLUSE
AND 4008.15  ; Reading completion (Exchange unit of lane 2)
TIM 0022 #0  ; ID writing start

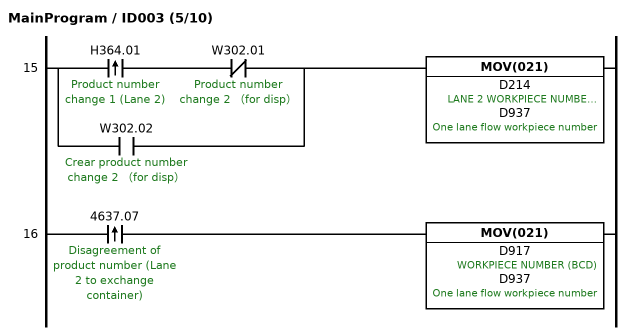
; rung 15
@LD H364.01  ; Product number change 1 (Lane 2)
ANDNOT W302.01  ; Product number change 2 （for disp）
OR W302.02  ; Crear product number change 2 （for disp）
MOV(021) D214 D937  ; LANE 2 WORKPIECE NUMBER DISPLAY, One lane flow workpiece number
; rung 16
@LD 4637.07  ; Disagreement of product number (Lane 2 to exchange container)
MOV(021) D917 D937  ; WORKPIECE NUMBER (BCD), One lane flow workpiece number

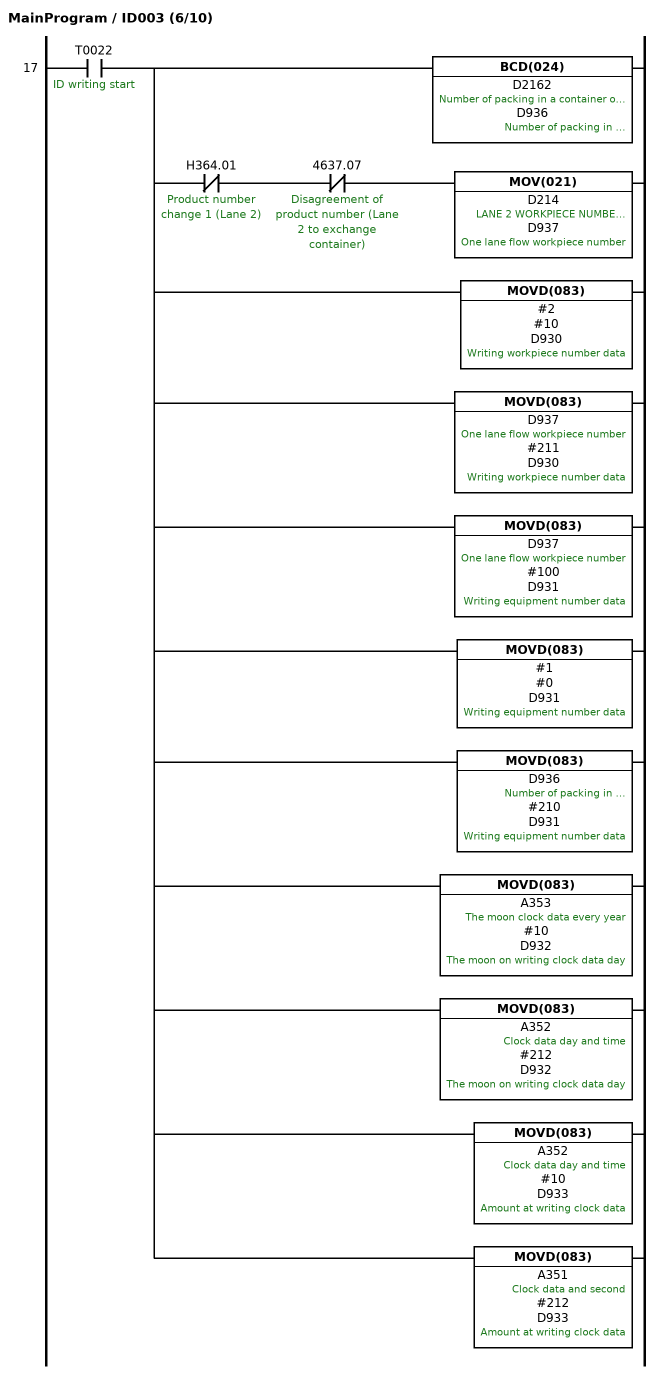
; rung 17
LD T0022  ; ID writing start
OUT TR0
BCD(024) D2162 D936  ; Number of packing in a container of lane 2 (exchange container)(BIN), Number of packing in a containrt(BCD)
ANDNOT H364.01  ; Product number change 1 (Lane 2)
ANDNOT 4637.07  ; Disagreement of product number (Lane 2 to exchange container)
MOV(021) D214 D937  ; LANE 2 WORKPIECE NUMBER DISPLAY, One lane flow workpiece number
LD TR0
MOVD(083) #2 #10 D930  ; Writing workpiece number data
MOVD(083) D937 #211 D930  ; One lane flow workpiece number, Writing workpiece number data
MOVD(083) D937 #100 D931  ; One lane flow workpiece number, Writing equipment number data
MOVD(083) #1 #0 D931  ; Writing equipment number data
MOVD(083) D936 #210 D931  ; Number of packing in a containrt(BCD), Writing equipment number data
MOVD(083) A353 #10 D932  ; The moon clock data every year, The moon on writing clock data day
MOVD(083) A352 #212 D932  ; Clock data day and time, The moon on writing clock data day
MOVD(083) A352 #10 D933  ; Clock data day and time, Amount at writing clock data
MOVD(083) A351 #212 D933  ; Clock data and second, Amount at writing clock data

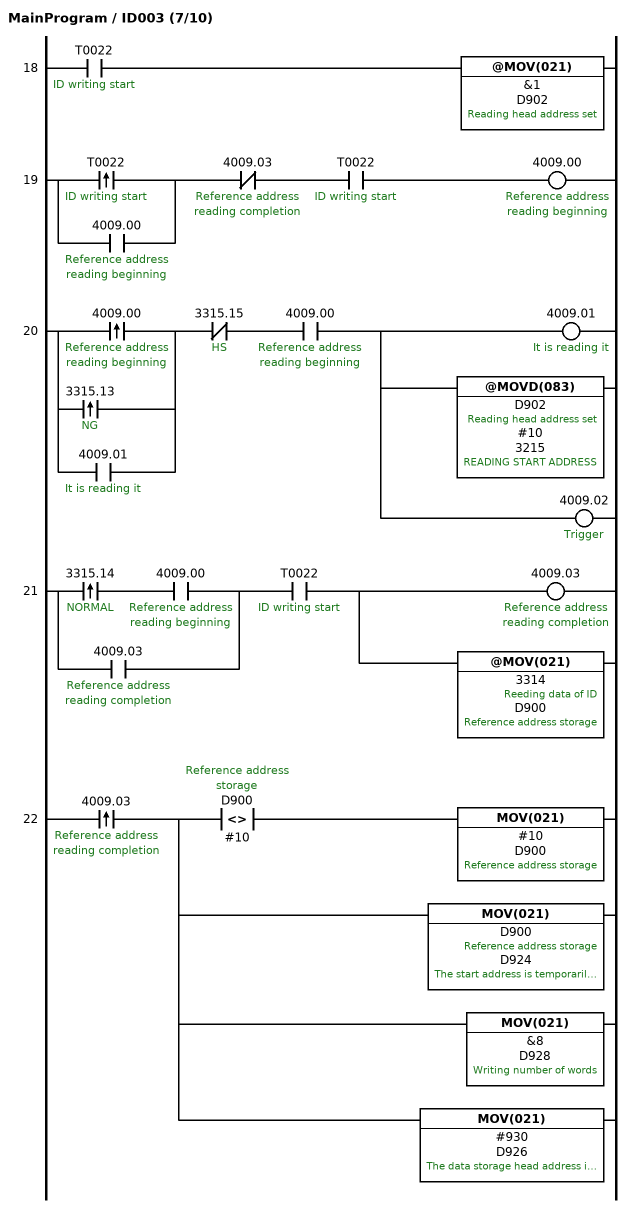
; rung 18
LD T0022  ; ID writing start
@MOV(021) &1 D902  ; Reading head address set
; rung 19
@LD T0022  ; ID writing start
OR 4009.00  ; Reference address reading beginning
ANDNOT 4009.03  ; Reference address reading completion
AND T0022  ; ID writing start
OUT 4009.00  ; Reference address reading beginning
; rung 20
@LD 4009.00  ; Reference address reading beginning
@OR 3315.13  ; NG
OR 4009.01  ; It is reading it
ANDNOT 3315.15  ; HS
AND 4009.00  ; Reference address reading beginning
OUT 4009.01  ; It is reading it
@MOVD(083) D902 #10 3215  ; Reading head address set, READING START ADDRESS
OUT 4009.02  ; Trigger
; rung 21
@LD 3315.14  ; NORMAL
AND 4009.00  ; Reference address reading beginning
OR 4009.03  ; Reference address reading completion
AND T0022  ; ID writing start
OUT 4009.03  ; Reference address reading completion
@MOV(021) 3314 D900  ; Reeding data of ID, Reference address storage
; rung 22
@LD 4009.03  ; Reference address reading completion
OUT TR0
AND<>(305) D900 #10  ; Reference address storage
MOV(021) #10 D900  ; Reference address storage
LD TR0
MOV(021) D900 D924  ; Reference address storage, The start address is temporarily memorized
MOV(021) &8 D928  ; Writing number of words
MOV(021) #930 D926  ; The data storage head address is memorized

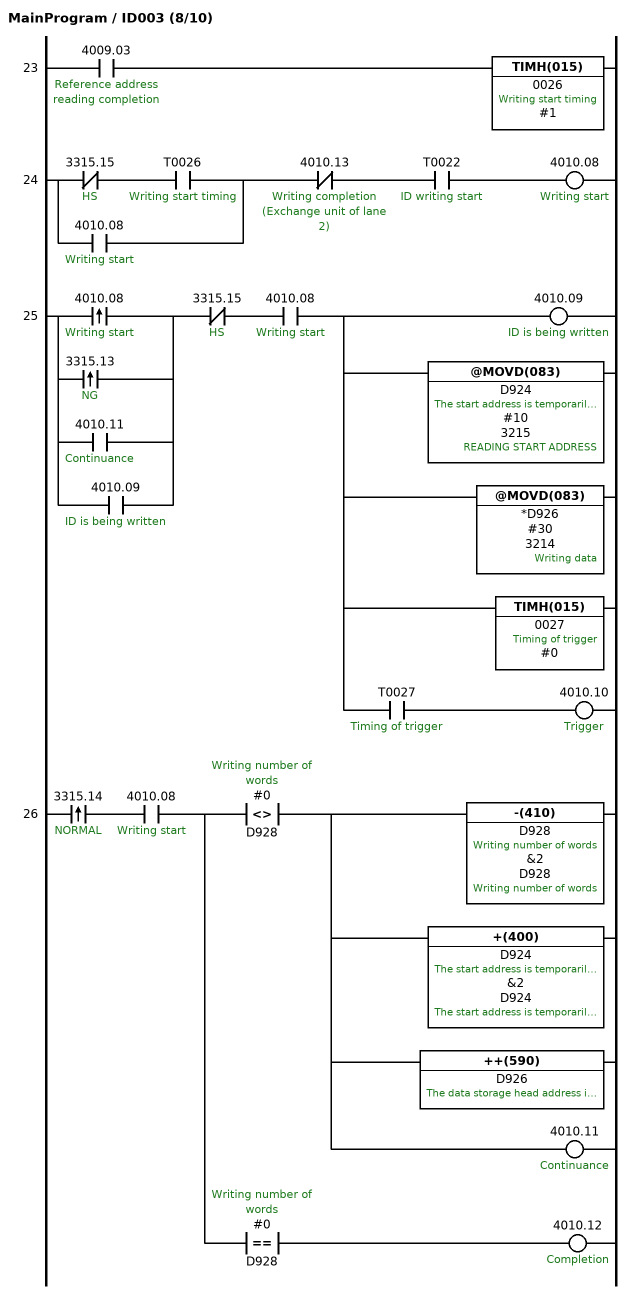
; rung 23
LD 4009.03  ; Reference address reading completion
TIMH(015) 0026 #1  ; Writing start timing
; rung 24
LDNOT 3315.15  ; HS
AND T0026  ; Writing start timing
OR 4010.08  ; Writing start
ANDNOT 4010.13  ; Writing completion (Exchange unit of lane 2)
AND T0022  ; ID writing start
OUT 4010.08  ; Writing start
; rung 25
@LD 4010.08  ; Writing start
@OR 3315.13  ; NG
OR 4010.11  ; Continuance
OR 4010.09  ; ID is being written
ANDNOT 3315.15  ; HS
AND 4010.08  ; Writing start
OUT 4010.09  ; ID is being written
@MOVD(083) D924 #10 3215  ; The start address is temporarily memorized, READING START ADDRESS
@MOVD(083) *D926 #30 3214  ; Writing data
TIMH(015) 0027 #0  ; Timing of trigger
AND T0027  ; Timing of trigger
OUT 4010.10  ; Trigger
; rung 26
@LD 3315.14  ; NORMAL
AND 4010.08  ; Writing start
OUT TR0
AND<>(305) #0 D928  ; Writing number of words
-(410) D928 &2 D928  ; Writing number of words
+(400) D924 &2 D924  ; The start address is temporarily memorized
++(590) D926  ; The data storage head address is memorized
OUT 4010.11  ; Continuance
LD TR0
AND=(300) #0 D928  ; Writing number of words
OUT 4010.12  ; Completion

